// TIA Portal V17 export
// export: Created 2022-07-20T07:02:31.9487711Z, ExportSetting WithDefaults, DisplayName Totally Integrated Automation Portal, DisplayVersion V17, DisplayName TIA Portal Openness, DisplayVersion V17, DisplayName TIA Portal Version Control Interface, DisplayVersion V17, DisplayName SINAMICS Startdrive Advanced, DisplayVersion V17, DisplayName SINAMICS Startdrive G130, G150, S120, S150, SINAMICS MV, S210, DisplayVersion V17, DisplayName SINAMICS Startdrive G110M, G120, G120C, G120D, G120P, G115D, DisplayVersion V17, DisplayName STEP 7 Professional, DisplayVersion V17, DisplayName STEP 7 Safety, DisplayVersion V17, DisplayName WinCC Advanced, DisplayVersion V17
FUNCTION_BLOCK "FB11007_VerticalMotor"   // FB11007, LAD
{ S7_Optimized_Access := 'TRUE' }
VERSION : 0.1
// stored: AutoNumber false, IsIECCheckEnabled false, IsRetainMemResEnabled false, MemoryReserve 100, SetENOAutomatically false, UDAEnableTagReadback false
   VAR_INPUT
      Fault : Bool;
      Homed : Bool;
      Ready : Bool;
      ExePos { ExternalAccessible := 'False'; ExternalVisible := 'False'; ExternalWritable := 'False'} : Bool;
      ExeHome : Bool;
      PosSelection { ExternalAccessible := 'False'; ExternalVisible := 'False'; ExternalWritable := 'False'} : UInt;
      ExeReset { ExternalAccessible := 'False'; ExternalVisible := 'False'; ExternalWritable := 'False'} : Bool;
      ExeStop { ExternalAccessible := 'False'; ExternalVisible := 'False'; ExternalWritable := 'False'} : Bool;
      TimeMeasureDownAdjustement : UInt;
   END_VAR
   VAR_OUTPUT
      Start : Bool;
      AlarmReset : Bool;
      DoHoming : Bool;
      Stop : Bool;
      M0 : Bool;
      M1 : Bool;
      M2 : Bool;
      InPosition { ExternalAccessible := 'False'; ExternalVisible := 'False'; ExternalWritable := 'False'} : Bool;
      AxisHomed { ExternalAccessible := 'False'; ExternalVisible := 'False'; ExternalWritable := 'False'} : Bool;
      StandStill { ExternalAccessible := 'False'; ExternalVisible := 'False'; ExternalWritable := 'False'} : Bool;
      PositionSelected { ExternalAccessible := 'False'; ExternalVisible := 'False'; ExternalWritable := 'False'} : UInt;
      TimeToDown { ExternalAccessible := 'False'; ExternalVisible := 'False'; ExternalWritable := 'False'} : UInt;
      AxisError : Bool;
   END_VAR
   VAR
      MotorMovementManagementStateDiagram : Int;
      TON_TimeMeasureToDown { S7_SetPoint := 'True'} : TON_TIME;
      TON_PositionSelected { S7_SetPoint := 'True'} : TON_TIME;
      R_TRIG_Ready { S7_SetPoint := 'True'} : R_TRIG;
      R_TRIG_ExePos { S7_SetPoint := 'True'} : R_TRIG;
      R_TRIG_ExeHome { S7_SetPoint := 'True'} : R_TRIG;
      F_TRIG_Ready { S7_SetPoint := 'True'} : R_TRIG;
      statExePos { S7_SetPoint := 'True'} : Bool;
   END_VAR
   VAR CONSTANT
      MOTOR_MOVEMENT_WAIT : Int := 0;
      MOTOR_DO_HOMING : Int := 10;
      MOTOR_SELECT_POSITION : Int := 20;
      MOTOR_GO_TO_POSITION : Int := 30;
      MOTOR_MOVEMENT_DONE : Int := 50;
   END_VAR
BEGIN

REGION Network 1 (SCL): Comments
   //==========================================================================================
   // SIEMENS SAS      RC-FR DI FA APC
   //------------------------------------------------------------------------------------------
   // Restrictions:    TIA V16 and more
   // Requirements:    S7-1500 + MGI library
   // Functionality:   This function block manage a vertical motor
   //------------------------------------------------------------------------------------------
   // Change log table:
   // Version      Date        Expert in charge    Changes applied
   // 01.00.01     09.06.2020  RTO                 First released version
   //==========================================================================================
END_REGION

REGION Network 2 (SCL): First Scan
   IF "FirstScan" THEN
       // Interface
       #PositionSelected := 0;
       #AxisHomed := FALSE;
       #InPosition := FALSE;
       #StandStill := FALSE;

       // Command
       #statExePos := FALSE;

       // Output
       #M0 := FALSE;
       #M1 := FALSE;
       #M2 := FALSE;
       #Start := FALSE;
       #AlarmReset := FALSE;
       #DoHoming := FALSE;
       #Stop := FALSE;

       //State Diagram
       #MotorMovementManagementStateDiagram := #MOTOR_MOVEMENT_WAIT;
   END_IF;
END_REGION

REGION Network 3 (SCL): Edge Signal Management
   REGION EDGE SIGNALS
       #R_TRIG_ExeHome(CLK := #ExeHome);
       #R_TRIG_ExePos(CLK := #ExePos);
       #R_TRIG_Ready(CLK := #Ready);

       IF #R_TRIG_ExePos.Q THEN
           #statExePos := TRUE;
       END_IF;

       #F_TRIG_Ready(CLK := #Ready);
   END_REGION

   REGION TIMERS
       // Signals
       #TON_PositionSelected(IN := #MotorMovementManagementStateDiagram = #MOTOR_SELECT_POSITION,
                         PT := T#4ms);

       // Mesaure time to down
       IF #R_TRIG_Ready.Q AND #PositionSelected <> 0 THEN
           #TimeToDown := TIME_TO_UINT(#TON_TimeMeasureToDown.ET) + #TimeMeasureDownAdjustement;
       END_IF;

       #TON_TimeMeasureToDown(IN := NOT #Ready AND #PositionSelected <> 0,
                                  PT := T#1m);
   END_REGION
END_REGION

REGION Network 4 (SCL): Manage position selected
   // CASE #PosSelection OF
   //     0:
   //         #PositionSelected := 0;
   //         #M0 := FALSE;
   //         #M1 := FALSE;
   //         #M2 := FALSE;
   //     1:
   //         #PositionSelected := 1;
   //         #M0 := TRUE;
   //         #M1 := FALSE;
   //         #M2 := FALSE;
   //     2:
   //         #PositionSelected := 2;
   //         #M0 := FALSE;
   //         #M1 := TRUE;
   //         #M2 := FALSE;
   //     3:
   //         #PositionSelected := 3;
   //         #M0 := TRUE;
   //         #M1 := TRUE;
   //         #M2 := FALSE;
   //     4:
   //         #PositionSelected := 4;
   //         #M0 := FALSE;
   //         #M1 := FALSE;
   //         #M2 := TRUE;
   //     5:
   //         #PositionSelected := 5;
   //         #M0 := TRUE;
   //         #M1 := FALSE;
   //         #M2 := TRUE;
   //     6:
   //         #PositionSelected := 6;
   //         #M0 := FALSE;
   //         #M1 := TRUE;
   //         #M2 := TRUE;
   //     7:
   //         #PositionSelected := 7;
   //         #M0 := TRUE;
   //         #M1 := TRUE;
   //         #M2 := TRUE;
   // END_CASE;
END_REGION

REGION Network 5 (SCL): Manage command
   (* IF #R_TRIG_ExePos.Q THEN
       #statExePos := TRUE;
   ELSIF #F_TRIG_Ready.Q THEN
       #statExePos := FALSE;
   END_IF; *)
END_REGION

REGION Network 6 (SCL)
   CASE #MotorMovementManagementStateDiagram OF
       #MOTOR_MOVEMENT_WAIT:
           IF #R_TRIG_ExeHome.Q AND #Ready THEN
               #MotorMovementManagementStateDiagram := #MOTOR_DO_HOMING;
           ELSIF #statExePos AND #Ready THEN //  #R_TRIG_ExePos.Q 
               #InPosition := FALSE;
               #statExePos := FALSE;
               #MotorMovementManagementStateDiagram := #MOTOR_SELECT_POSITION; //#MOTOR_GO_TO_POSITION;
           END_IF;
       #MOTOR_DO_HOMING:
           #DoHoming := TRUE;
           IF NOT(#Ready) THEN
               #DoHoming := FALSE;
               #MotorMovementManagementStateDiagram := #MOTOR_MOVEMENT_DONE;
           END_IF;
       #MOTOR_SELECT_POSITION:
           IF #PosSelection = 0 THEN
               #PositionSelected := 0;
               #M0 := FALSE;
               #M1 := FALSE;
               #M2 := FALSE;
           ELSIF #PosSelection = 1 THEN
               #PositionSelected := 1;
               #M0 := TRUE;
               #M1 := FALSE;
               #M2 := FALSE;
           ELSIF #PosSelection = 2 THEN
               #PositionSelected := 2;
               #M0 := FALSE;
               #M1 := TRUE;
               #M2 := FALSE;
           ELSIF #PosSelection = 3 THEN
               #PositionSelected := 3;
               #M0 := TRUE;
               #M1 := TRUE;
               #M2 := FALSE;
           ELSIF #PosSelection = 4 THEN
               #PositionSelected := 4;
               #M0 := FALSE;
               #M1 := FALSE;
               #M2 := TRUE;
           ELSIF #PosSelection = 5 THEN
               #PositionSelected := 5;
               #M0 := TRUE;
               #M1 := FALSE;
               #M2 := TRUE;
           ELSIF #PosSelection = 6 THEN
               #PositionSelected := 6;
               #M0 := FALSE;
               #M1 := TRUE;
               #M2 := TRUE;
           ELSIF #PosSelection = 7 THEN
               #PositionSelected := 7;
               #M0 := TRUE;
               #M1 := TRUE;
               #M2 := TRUE;
           END_IF;
           IF #TON_PositionSelected.Q THEN
               RESET_TIMER(#TON_PositionSelected);
               #MotorMovementManagementStateDiagram := #MOTOR_GO_TO_POSITION;
           END_IF;
       #MOTOR_GO_TO_POSITION:
           #Start := TRUE;
           IF NOT (#Ready) THEN
               #Start := FALSE;
           ELSIF #R_TRIG_Ready.Q THEN
               #M0 := FALSE;
               #M1 := FALSE;
               #M2 := FALSE;
               #Start := FALSE;
               #InPosition := TRUE;
               #MotorMovementManagementStateDiagram := #MOTOR_MOVEMENT_DONE;
           END_IF;
       #MOTOR_MOVEMENT_DONE:
           #MotorMovementManagementStateDiagram := #MOTOR_MOVEMENT_WAIT;
   END_CASE;
END_REGION

REGION Network 7 (SCL): Manage Output
   (* IF #statExePos AND #TON_PositionSelected.Q AND #Ready THEN
       #Start := TRUE;
   ELSIF NOT #Ready THEN
       #Start := FALSE;
   END_IF;

   IF #R_TRIG_ExeHome.Q AND #Ready THEN
       #DoHoming := TRUE;
   ELSIF #F_TRIG_Ready.Q THEN
       #DoHoming := FALSE;
   END_IF; *)

   #Stop := #ExeStop;
   #AlarmReset := #ExeReset;
END_REGION

REGION Network 8 (SCL): Manage state
   #AxisHomed := #Homed;

   (* IF #R_TRIG_Ready.Q THEN
       #InPosition := TRUE;
   ELSIF #R_TRIG_ExePos.Q THEN
       #InPosition := FALSE;
   END_IF;
   *)
   #StandStill := #Ready;
END_REGION

REGION Network 9 (SCL): Manage error
   #AxisError := NOT #Fault;
END_REGION
END_FUNCTION_BLOCK
